// TIA Portal V17 export
// export: Created 2025-03-05T07:59:56.6172483Z, ExportSetting WithDefaults, DisplayName Totally Integrated Automation Portal, DisplayVersion V17 Update 8, DisplayName TIA Portal Openness, DisplayVersion V17 Update 8, DisplayName TIA Portal Version Control Interface, DisplayVersion V17, DisplayName SINAMICS Startdrive Advanced, DisplayVersion V17 SP2, DisplayName SINAMICS Startdrive G110M, G120, G120C, G120D, G120P, G115D, DisplayVersion V17 SP2, DisplayName SINAMICS Startdrive G130, G150, S120, S150, SINAMICS MV, S210, DisplayVersion V17 SP2, DisplayName STEP 7 Professional, DisplayVersion V17 Update 8, DisplayName SINUMERIK ONE STEP 7 Toolbox, DisplayVersion V17 Update 12, DisplayName SINUMERIK 840D sl STEP 7 Toolbox, DisplayVersion V17 Update 12, DisplayName STEP 7 Safety, DisplayVersion V17 Update 6, DisplayName WinCC Advanced, DisplayVersion V17 Update 8
DATA_BLOCK "DB427_VARIABLE_ALARM"   // DB427
{ S7_Optimized_Access := 'FALSE'; DB_Accessible_From_OPC_UA := 'FALSE' }
AUTHOR : ETXETAR
VERSION : 1.0
// stored: AutoNumber false, DBAccessibleFromOPCUA false, DBAccessibleFromWebserver true, IsOnlyStoredInLoadMemory false, IsWriteProtectedInAS false
   VAR RETAIN
      FAULTS : Struct
         TRIGGER_BIT : Array[0..15] of Bool;
         DATA_FOR_VAR_FAULT : Array[0..15] of Struct
            FAULT_NUMBER : Word;
            EVALUATION_BITS : Word;
            PARAMETER_1 : Word;
            PARAMETER_2 : Word;
            PARAMETER_3 : Word;
            PARAMETER_4 : Word;
         END_STRUCT;
         STA_01R : Struct
            FAULT_NUMBER : Word;
            PARAMETER_1 : Word;
            PARAMETER_2 : Word;
            PARAMETER_3 : Word;
            PARAMETER_4 : Word;
            MEMORY_FAULT_SET : Int;
         END_STRUCT;
         STA_01L : Struct
            FAULT_NUMBER : Word;
            PARAMETER_1 : Word;
            PARAMETER_2 : Word;
            PARAMETER_3 : Word;
            PARAMETER_4 : Word;
            MEMORY_FAULT_SET : Int;
         END_STRUCT;
      END_STRUCT;
   END_VAR
BEGIN
END_DATA_BLOCK
